(* Logix 5000 project; controller SinglePumpTest vendor 1 type 14 code 196 rev 33.11; software revision 33.00 *)

TASK MainTask (continuous, watchdog 500 ms) : MainProgram

MODULES
   Local : vendor 1 type 14 code 196 (5069 0, rev 33.11)
      VMP_00 : vendor 1449 type 43 code 17 (Ethernet 192.168.2.130, rev 1.4, StandardDataDriven RPI 500 ms)
      IN : 5069-IB16 (5069 2, rev 2.1, StandardDataDriven RPI 5 ms)   // Input Module
      OUT : vendor 1 type 7 code 396 (5069 1, rev 2.1, StandardDataDriven RPI 5 ms)   // Output Module
END_MODULES

TYPE STRING_12 :
STRUCT
   LEN : DINT;
   DATA : SINT[12];
END_STRUCT
END_TYPE

TYPE STRING_24 :
STRUCT
   LEN : DINT;
   DATA : SINT[24];
END_STRUCT
END_TYPE

TYPE VMP_Input :   // Data received from the Pump
STRUCT
   vmpStatus : DINT;   // Bits indicating the status
   vmpStatus_Ready : BOOL;   // Pump is ready to run
   vmpStatus_Running : BOOL;   // Pump is running.
   vmpStatus_Abort : BOOL;   // Pump is in an Abort state
   vmpStatus_Direction : BOOL;   // Turning counter clockwise
   vmpStatus_ContinuousRun : BOOL;   // In continuous run mode
   vmpStatus_MotorRunning : BOOL;   // One of the motors is running
   vmpFaults : DINT;   // Faults as a bit mask
   vmpFaults_DispenseMotor : BOOL;   // Dispense Motor
   vmpFaults_AdjustMotor : BOOL;   // Adjustmemt Motor
   SpareBits : DINT;   // Spara Data bits
   currentProgram : DINT;   // Current selected program
   revolutions : DINT;   // Number of revolutions
   SpareDInt1 : DINT;   // Spare data
   SpareDInt2 : DINT;   // Spare data
   SpareDInt3 : DINT;   // Spare data
   SpareDInt4 : DINT;   // Spare data
   volume : REAL;   // Current volume
   SpareReal1 : REAL;   // Spare data
   SpareReal2 : REAL;   // Spare data
   SpareReal3 : REAL;   // Spare data
   SpareReal4 : REAL;   // Spare data
END_STRUCT
END_TYPE

TYPE VMP_Output :   // Data sent to the pump
STRUCT
   plcCmd : DINT;   // Pump commands as bit fields
   plcCmd_Ready : BOOL;   // Ok to run pump
   plcCmd_Start : BOOL;   // Start the pump
   plcCmd_Abort : BOOL;   // Abort Running program
   plcCmd_Direction : BOOL;   // Turning counter clockwise
   plcCmd_ContinuousRun : BOOL;   // Run continuously
   plcCmd_SetMaxShotSize : BOOL;   // Set volume to max size
   Spare : DINT;   // Spare bits
   currentProgram : DINT;   // Proram number to run
   revolutions : DINT;   // Number of revolutions to turn
   Spare_1 : DINT;   // Spare data
   Spare_2 : DINT;   // Spare data
   Spare_3 : DINT;   // Spare data
   Spare_4 : DINT;   // Spare data
   volume : REAL;   // Set volume size
   SpareReal_1 : REAL;   // Spare data
   SpareReal_2 : REAL;   // Spare data
   SpareReal_3 : REAL;   // Spare data
   SpareReal_4 : REAL;   // Spare data
END_STRUCT
END_TYPE

TYPE VMP_Program :   // Program Parameters
STRUCT
   Current_Program : DINT;   // Currently Selected Program
   Direction : DINT;   // Rotational direction of the pump motor.
   Pull_Back : DINT;   // Percentage rotation to reverse the pump after a shot. E.g. suck back.
   Initial_RPM : DINT;   // Initial speed of the pump.
   RPM : DINT;   // Speed of the pump after initial RPM
   Final_RPM : DINT;   // Final speed of the pump after RPM.
   Fine_Adjust : DINT;   // 1=Increment, 0=Clear, -1=Decrement fine adjust.
   Set_Shot : DINT;   // Reset size to zero then to current program setting.
   Acceleration : DINT;   // Set speed of acceleration for initial RPM.
   Deceleration : DINT;   // Set speed of deceleration for final RPM.
   Loop_Cycles : DINT;   // Number of times to run the linked program.
   Linked_Program : DINT;   // -1=Disabled, 0 to 49 next program to run.
   Linked_Time_Delay : DINT;   // Number of seconds to wait before running the linked program.
   Motor_Current : DINT;   // Percentage current used to drive the motor.
   Continuous_Run : DINT;   // 0=Normal Mode, 1=Continuous Run Mode
   Revolutions : DINT;   // Number of revolutions to turn the pump head.
   Approx_Time : DINT;   // Approximate time in mill-seconds for a dispense time.
   Volume : REAL;   // Shot Volume
   Program_Name : STRING;   // Name of the current program.
END_STRUCT
END_TYPE

TYPE VMP_Setup :
STRUCT
   CosType : INT;   // CosType
   ClassId : INT;   // ClassId
   Instance : INT;   // Instance
   Attribute : INT;   // Attribute
   CfgVersion : INT;   // CfgVersion
   CfgLength : INT;   // CfgLength
   NumberOfHeads : SINT;   // NumberOfHeads
   PumpType : SINT;   // PumpType
   PumpNumber : SINT;   // PumpNumber
   SpareByte1 : SINT;   // SpareByte1
   AdjustStepmode : INT;   // AdjustStepmode
   ZinchRpm : INT;   // ZinchRpm
   Baud : INT;   // Baud
   ExtraSteps : INT;   // ExtraSteps
   SpareInt1 : INT;   // SpareInt1
   SpareInt2 : INT;   // SpareInt2
   ReadyInterlock : BOOL;   // ReadyInterlock
   EthernetRunReady : BOOL;   // EthernetRunReady
   DchpEnabled : BOOL;   // DchpEnabled
   BoreInCm : BOOL;   // BoreInCm
   IoStartFallingEdge : BOOL;   // IoStartFallingEdge
   FullDuplexRs485 : BOOL;   // FullDuplexRs485
   Spare1_6 : BOOL;   // Spare1_6
   Spare1_7 : BOOL;   // Spare1_7
   Spare1_8 : BOOL;   // Spare1_8
   Spare1_9 : BOOL;   // Spare1_9
   Spare1_10 : BOOL;   // Spare1_10
   Spare1_11 : BOOL;   // Spare1_11
   Spare1_12 : BOOL;   // Spare1_12
   Spare1_13 : BOOL;   // Spare1_13
   Spare1_14 : BOOL;   // Spare1_14
   Spare1_15 : BOOL;   // Spare1_15
   Spare1_16 : BOOL;   // Spare1_16
   Spare1_17 : BOOL;   // Spare1_17
   Spare1_18 : BOOL;   // Spare1_18
   Spare1_19 : BOOL;   // Spare1_19
   Spare1_20 : BOOL;   // Spare1_20
   Spare1_21 : BOOL;   // Spare1_21
   Spare1_22 : BOOL;   // Spare1_22
   Spare1_23 : BOOL;   // Spare1_23
   IsServo : BOOL;   // IsServo
   OkToResetDevice : BOOL;   // OkToResetDevice
   Spare1_26 : BOOL;   // Spare1_26
   Spare1_27 : BOOL;   // Spare1_27
   Spare1_28 : BOOL;   // Spare1_28
   Spare1_29 : BOOL;   // Spare1_29
   Spare1_30 : BOOL;   // Spare1_30
   Spare1_31 : BOOL;   // Spare1_31
   FirmwareRev : DINT;   // FirmwareRev
   Bore : DINT;   // Bore
   OffsetValue : DINT;   // OffsetValue
   FlashWriteCnt : DINT;   // FlashWriteCnt
   FaultDispenseSensorCnt : DINT;   // FaultDispenseSensorCnt
   FaultDispenseMotorCnt : DINT;   // FaultDispenseMotorCnt
   FaultAdjustSensorCnt : DINT;   // FaultAdjustSensorCnt
   FaultAdjustMotorCnt : DINT;   // FaultAdjustMotorCnt
   SpareDInt1 : DINT;   // SpareDInt1
   SpareDint2 : DINT;   // SpareDint2
   SerialNumber : STRING_16;   // SerialNumber
   IpAddress : STRING_16;   // IpAddress
   IpNetmask : STRING_16;   // IpNetmask
   IpGateway : STRING_16;   // IpGateway
   MacAddress : STRING_24;   // MacAddress
   ModelNumber : STRING_24;   // ModelNumber
   OptionsAndFittings : STRING_24;   // OptionsAndFittings
   SccsRevDate : STRING_24;   // SccsRevDate
   SccsRev : STRING_12;   // SccsRev
   SccsRevRange : STRING_24;   // SccsRevRange
END_STRUCT
END_TYPE

PROGRAM MainProgram   (* main routine MainRoutine *)
VAR
   Run : BOOL;
   Run_ONS : BOOL;
END_VAR

ROUTINE MainRoutine   (* ladder *)
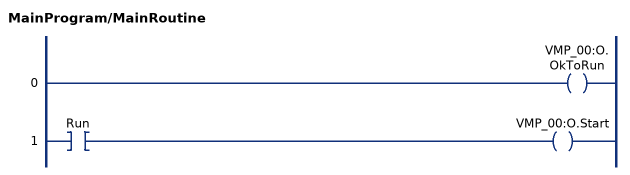
   0: OTE(VMP_00:O.OkToRun);
   1: XIC(Run)OTE(VMP_00:O.Start);
END_ROUTINE
END_PROGRAM
